TYPE commCommandPos EXTENDS commCommandBase :
STRUCT
	controlWord:DWORD; //16,17 , bit0, true=abs
	coordinate:DINT; //18,19 , in 0.001mm
END_STRUCT
END_TYPE

(* stored: Version 1.1.0.1, ProductVersion 3.1.4022.10
   DUT commCommandPos: Id {8f368442-c415-42b2-b751-673ee70c0436} *)
